// LS Electric XG5000 project: 16-04-1
// PLC NewPLC
// module base 0 slot 0: 입출력 모듈:XBC-DN/DP14E (DC 24V 입력 8점, 트랜지스터 출력 6점)

PROGRAM NewProgram (task: 스캔 프로그램)

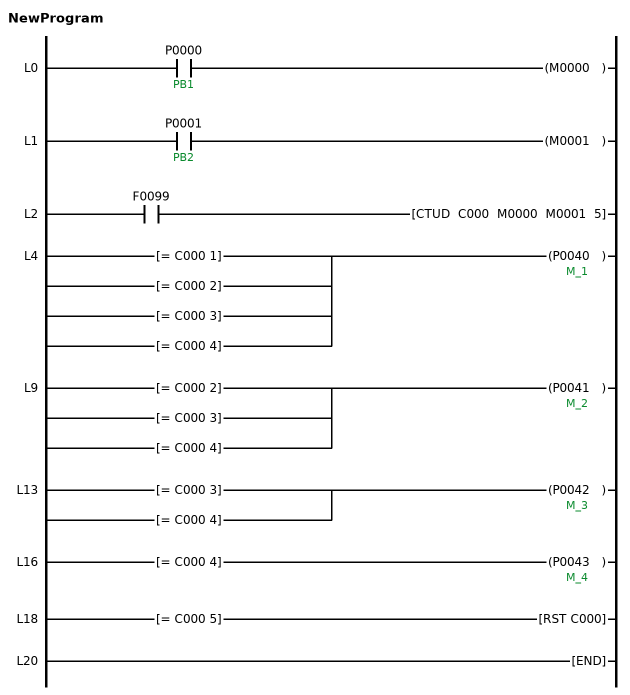
; L0
LOAD      P0000	// PB1
OUT       M0000
; L1
LOAD      P0001	// PB2
OUT       M0001
; L2
LOAD      F0099
CTUD      C000 M0000 M0001 5
; L4
LOAD=     C000 1
OR=       C000 2
OR=       C000 3
OR=       C000 4
OUT       P0040	// M_1
; L9
LOAD=     C000 2
OR=       C000 3
OR=       C000 4
OUT       P0041	// M_2
; L13
LOAD=     C000 3
OR=       C000 4
OUT       P0042	// M_3
; L16
LOAD=     C000 4
OUT       P0043	// M_4
; L18
LOAD=     C000 5
RST       C000
; L20
END